Staubli VAL3: delEvent.pgx

program delEvent(num x_nIndex (dimensions=1))
begin
  // delete the item
  if size(pEdit.iEvent)>1
    delete(pEdit.iEvent[x_nIndex])
  else
    pEdit.iEvent.sType=""
    pEdit.iEvent.sData=""
  endIf
end
